PROGRAM Z_CP

VAR
	rOutAnalogVelPump: REAL;
	DD: REAL;
END_VAR

//Activar Bomba

Mc._09_CPUMP.b450_CircPump.xRUN:= _00_CIRC_PUMP.Marcha.Run;


//Velocidad

rOutAnalogVelPump	:= Canvi_Escala(In:= mc._08_CIRC.rSP_SpeedPumpC,
									In_Min:=0,
									In_Max:=100,
									Out_Min:= 0,
									Out_Max:= 32767);
									
DD:=	rOutAnalogVelPump;

END_PROGRAM

(* stored: Version 1.1.0.1, ProductVersion 3.1.4024.10
   POU Z_CP: Id {c5d69aa4-0f0e-4233-909e-503d0ba27b8e}, SpecialFunc None *)
